// TIA Portal V19 export
TYPE "TAx_Speed_Alarms"
// stored: Access Published
   STRUCT
      TOAxis : Bool;   // Alarm in technology object
      MCFunction : Bool;   // Alarm of MC function
      Drive : Bool;   // Alarm in the drive
   END_STRUCT;
END_TYPE
